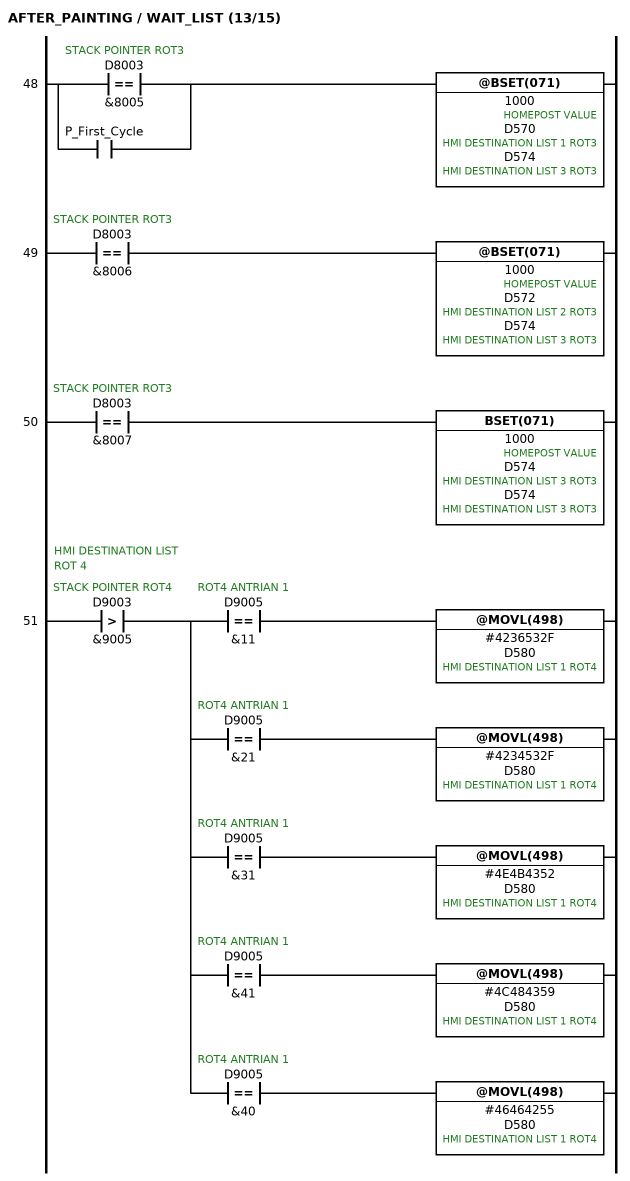
; [picture p96: AFTER_PAINTING / WAIT_LIST, rungs 48-51]
; rung 48
LD=(300) D8003 &8005  ; STACK POINTER ROT3
OR P_First_Cycle
@BSET(071) 1000 D570 D574  ; HOMEPOST VALUE, HMI DESTINATION LIST 1 ROT3, HMI DESTINATION LIST 3 ROT3
; rung 49
LD=(300) D8003 &8006  ; STACK POINTER ROT3
@BSET(071) 1000 D572 D574  ; HOMEPOST VALUE, HMI DESTINATION LIST 2 ROT3, HMI DESTINATION LIST 3 ROT3
; rung 50
LD=(300) D8003 &8007  ; STACK POINTER ROT3
BSET(071) 1000 D574 D574  ; HOMEPOST VALUE, HMI DESTINATION LIST 3 ROT3
; rung 51: HMI DESTINATION LIST / ROT 4
LD>(320) D9003 &9005  ; STACK POINTER ROT4
OUT TR0
AND=(300) D9005 &11  ; ROT4 ANTRIAN 1
@MOVL(498) #4236532F D580  ; HMI DESTINATION LIST 1 ROT4
LD TR0
AND=(300) D9005 &21  ; ROT4 ANTRIAN 1
@MOVL(498) #4234532F D580  ; HMI DESTINATION LIST 1 ROT4
LD TR0
AND=(300) D9005 &31  ; ROT4 ANTRIAN 1
@MOVL(498) #4E4B4352 D580  ; HMI DESTINATION LIST 1 ROT4
LD TR0
AND=(300) D9005 &41  ; ROT4 ANTRIAN 1
@MOVL(498) #4C484359 D580  ; HMI DESTINATION LIST 1 ROT4
LD TR0
AND=(300) D9005 &40  ; ROT4 ANTRIAN 1
@MOVL(498) #46464255 D580  ; HMI DESTINATION LIST 1 ROT4

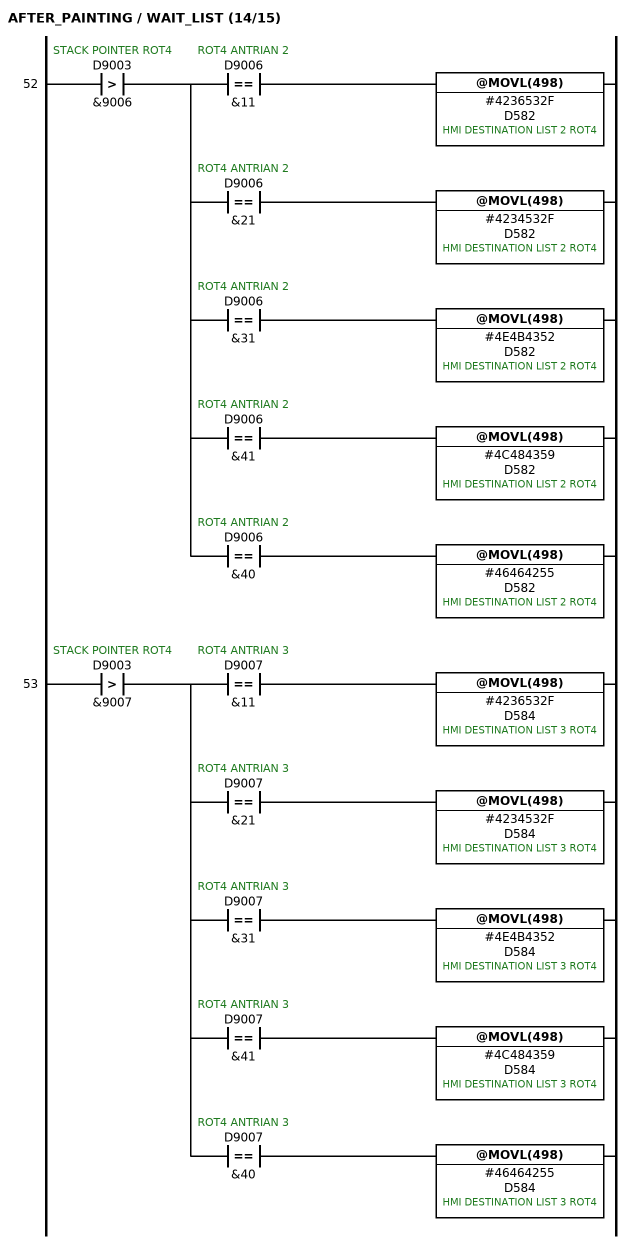
; rung 52
LD>(320) D9003 &9006  ; STACK POINTER ROT4
OUT TR0
AND=(300) D9006 &11  ; ROT4 ANTRIAN 2
@MOVL(498) #4236532F D582  ; HMI DESTINATION LIST 2 ROT4
LD TR0
AND=(300) D9006 &21  ; ROT4 ANTRIAN 2
@MOVL(498) #4234532F D582  ; HMI DESTINATION LIST 2 ROT4
LD TR0
AND=(300) D9006 &31  ; ROT4 ANTRIAN 2
@MOVL(498) #4E4B4352 D582  ; HMI DESTINATION LIST 2 ROT4
LD TR0
AND=(300) D9006 &41  ; ROT4 ANTRIAN 2
@MOVL(498) #4C484359 D582  ; HMI DESTINATION LIST 2 ROT4
LD TR0
AND=(300) D9006 &40  ; ROT4 ANTRIAN 2
@MOVL(498) #46464255 D582  ; HMI DESTINATION LIST 2 ROT4
; rung 53
LD>(320) D9003 &9007  ; STACK POINTER ROT4
OUT TR0
AND=(300) D9007 &11  ; ROT4 ANTRIAN 3
@MOVL(498) #4236532F D584  ; HMI DESTINATION LIST 3 ROT4
LD TR0
AND=(300) D9007 &21  ; ROT4 ANTRIAN 3
@MOVL(498) #4234532F D584  ; HMI DESTINATION LIST 3 ROT4
LD TR0
AND=(300) D9007 &31  ; ROT4 ANTRIAN 3
@MOVL(498) #4E4B4352 D584  ; HMI DESTINATION LIST 3 ROT4
LD TR0
AND=(300) D9007 &41  ; ROT4 ANTRIAN 3
@MOVL(498) #4C484359 D584  ; HMI DESTINATION LIST 3 ROT4
LD TR0
AND=(300) D9007 &40  ; ROT4 ANTRIAN 3
@MOVL(498) #46464255 D584  ; HMI DESTINATION LIST 3 ROT4

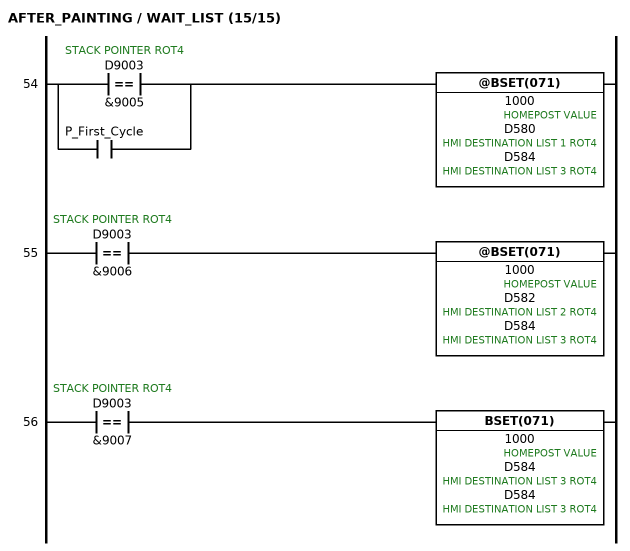
; rung 54
LD=(300) D9003 &9005  ; STACK POINTER ROT4
OR P_First_Cycle
@BSET(071) 1000 D580 D584  ; HOMEPOST VALUE, HMI DESTINATION LIST 1 ROT4, HMI DESTINATION LIST 3 ROT4
; rung 55
LD=(300) D9003 &9006  ; STACK POINTER ROT4
@BSET(071) 1000 D582 D584  ; HOMEPOST VALUE, HMI DESTINATION LIST 2 ROT4, HMI DESTINATION LIST 3 ROT4
; rung 56
LD=(300) D9003 &9007  ; STACK POINTER ROT4
BSET(071) 1000 D584 D584  ; HOMEPOST VALUE, HMI DESTINATION LIST 3 ROT4

### Section END
; rung 0
END(001)

## Function block MANUAL_ROTARY
VAR_INPUT
  PB_HMI_TURN : BOOL;
  PB_HMI_STRAIGHT : BOOL;
  PB_EXECUTE : BOOL;
  RS_PINLOCK_UP : BOOL;
  RS_PINLOCK_DOWN : BOOL;
  LS_STRAIGHT : BOOL;
  LS_TURN : BOOL;
  HOMEPOST_STRAIGHT : BOOL;
  HOMEPOST_RESET : BOOL;
END_VAR
VAR_OUTPUT
  MOTOR_FWD : BOOL;
  MOTOR_RVS : BOOL;
  PINLOCK_UP : BOOL;
  PINLOCK_DOWN : BOOL;
END_VAR
VAR
  MOTOR_RVS_MANUAL : BOOL;
  MOTOR_RVS_HOMEPOST : BOOL;
  PINLOCK_UP_STRAIGHT : BOOL;
  PINLOCK_UP_TURN : BOOL;
  PINLOCK_DOWN_STRAIGHT : BOOL;
  PINLOCK_DOWN_TURN : BOOL;
  PINLOCK_UP_HOMEPOST : BOOL;
  PINLOCK_DOWN_HOMEPOST : BOOL;
END_VAR

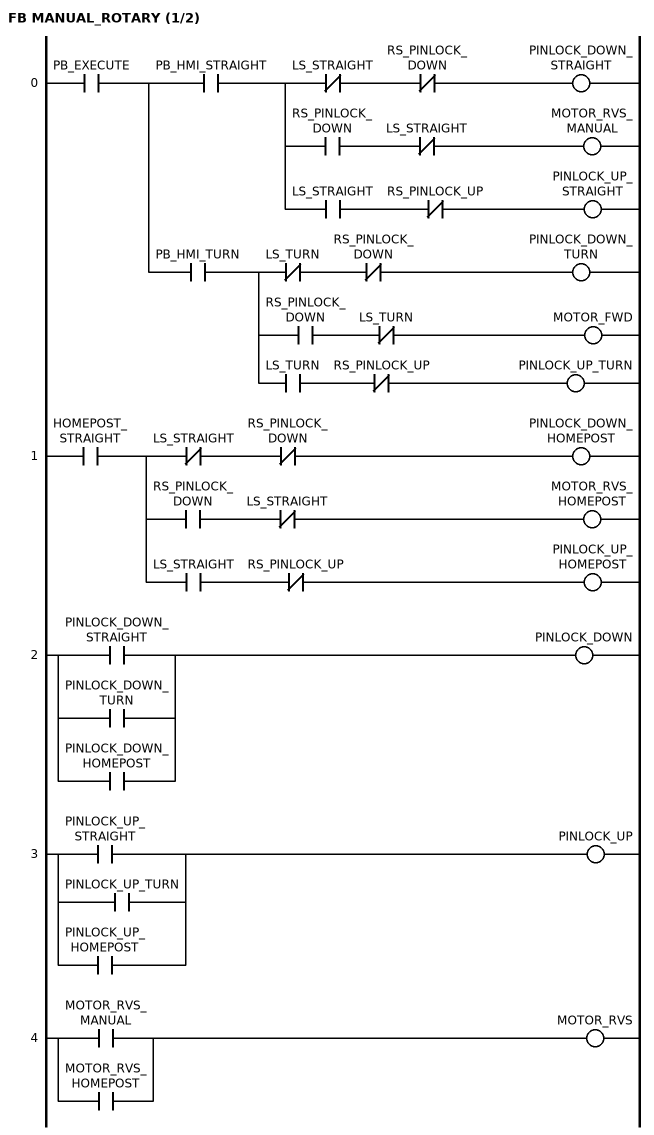
; rung 0
LD PB_EXECUTE
OUT TR0
AND PB_HMI_STRAIGHT
OUT TR1
ANDNOT LS_STRAIGHT
ANDNOT RS_PINLOCK_DOWN
OUT PINLOCK_DOWN_STRAIGHT
LD TR1
AND RS_PINLOCK_DOWN
ANDNOT LS_STRAIGHT
OUT MOTOR_RVS_MANUAL
LD TR1
AND LS_STRAIGHT
ANDNOT RS_PINLOCK_UP
OUT PINLOCK_UP_STRAIGHT
LD TR0
AND PB_HMI_TURN
OUT TR2
ANDNOT LS_TURN
ANDNOT RS_PINLOCK_DOWN
OUT PINLOCK_DOWN_TURN
LD TR2
AND RS_PINLOCK_DOWN
ANDNOT LS_TURN
OUT MOTOR_FWD
LD TR2
AND LS_TURN
ANDNOT RS_PINLOCK_UP
OUT PINLOCK_UP_TURN
; rung 1
LD HOMEPOST_STRAIGHT
OUT TR0
ANDNOT LS_STRAIGHT
ANDNOT RS_PINLOCK_DOWN
OUT PINLOCK_DOWN_HOMEPOST
LD TR0
AND RS_PINLOCK_DOWN
ANDNOT LS_STRAIGHT
OUT MOTOR_RVS_HOMEPOST
LD TR0
AND LS_STRAIGHT
ANDNOT RS_PINLOCK_UP
OUT PINLOCK_UP_HOMEPOST
; rung 2
LD PINLOCK_DOWN_STRAIGHT
OR PINLOCK_DOWN_TURN
OR PINLOCK_DOWN_HOMEPOST
OUT PINLOCK_DOWN
; rung 3
LD PINLOCK_UP_STRAIGHT
OR PINLOCK_UP_TURN
OR PINLOCK_UP_HOMEPOST
OUT PINLOCK_UP
; rung 4
LD MOTOR_RVS_MANUAL
OR MOTOR_RVS_HOMEPOST
OUT MOTOR_RVS

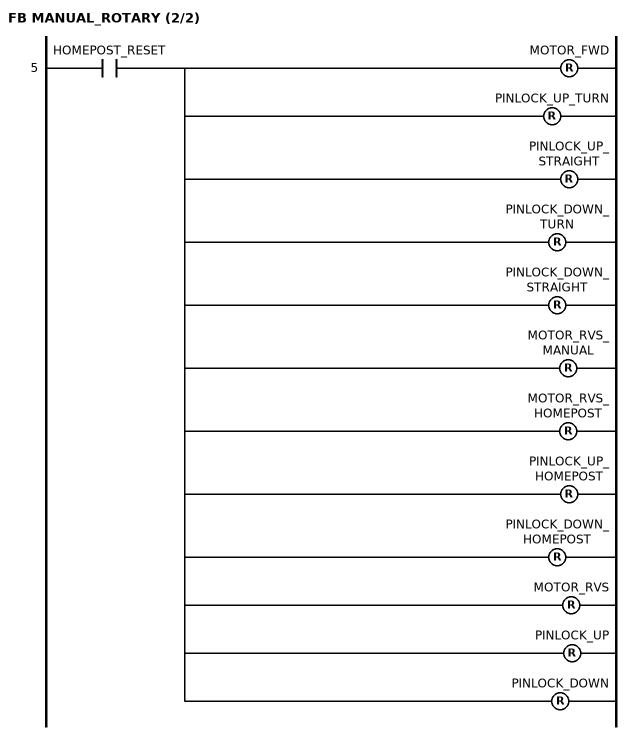
; rung 5
LD HOMEPOST_RESET
RSET MOTOR_FWD
RSET PINLOCK_UP_TURN
RSET PINLOCK_UP_STRAIGHT
RSET PINLOCK_DOWN_TURN
RSET PINLOCK_DOWN_STRAIGHT
RSET MOTOR_RVS_MANUAL
RSET MOTOR_RVS_HOMEPOST
RSET PINLOCK_UP_HOMEPOST
RSET PINLOCK_DOWN_HOMEPOST
RSET MOTOR_RVS
RSET PINLOCK_UP
RSET PINLOCK_DOWN

## Function block RFID_SEQUENCE
VAR_INPUT
  PB_SAVE : BOOL;
  AUTO_SEQ_ON : BOOL;
  INPUT_DATA : UINT;
  PH_OUT : BOOL;
  MANUAL_MODE : BOOL;
  PB_CLEAR_MEMORY : BOOL;
  PB_ENABLE_READER : BOOL;
  OUT_HMI_DISPLAY_NO_RFID : UDINT;
  STACK_LOC : UINT;
  REDUDANCY_ACCEPTED : BOOL;
  HOMEPOST_RESET : BOOL;
END_VAR
VAR_OUTPUT
  RFID_CONFIRM_MATCH : BOOL;
  DISPLAY_TEACH_RFID : UDINT;
  ALARM_RFID_NOT_DETECT : BOOL;
  DATA_REDUDANCY : BOOL;
  RETAIN MEMORY_1 : UDINT;
  RETAIN MEMORY_2 : UDINT;
  RETAIN MEMORY_3 : UDINT;
  RETAIN MEMORY_4 : UDINT;
  RETAIN MEMORY_5 : UDINT;
  RETAIN MEMORY_6 : UDINT;
  RETAIN MEMORY_7 : UDINT;
  RETAIN MEMORY_8 : UDINT;
  RETAIN MEMORY_9 : UDINT;
  RETAIN MEMORY_10 : UDINT;
  RETAIN MEMORY_11 : UDINT;
  RETAIN MEMORY_12 : UDINT;
  RETAIN MEMORY_13 : UDINT;
  RETAIN MEMORY_14 : UDINT;
  RETAIN MEMORY_15 : UDINT;
  RETAIN MEMORY_16 : UDINT;
  RETAIN MEMORY_17 : UDINT;
  RETAIN MEMORY_18 : UDINT;
  RETAIN MEMORY_19 : UDINT;
  RETAIN MEMORY_20 : UDINT;
  RETAIN MEMORY_21 : UDINT;
  RETAIN MEMORY_22 : UDINT;
  RETAIN MEMORY_23 : UDINT;
  RETAIN MEMORY_24 : UDINT;
  RETAIN MEMORY_25 : UDINT;
  RETAIN MEMORY_26 : UDINT;
  RETAIN MEMORY_27 : UDINT;
  RETAIN MEMORY_28 : UDINT;
  RETAIN MEMORY_29 : UDINT;
  RETAIN MEMORY_30 : UDINT;
  RETAIN MEMORY_31 : UDINT;
  RETAIN MEMORY_32 : UDINT;
  RETAIN MEMORY_33 : UDINT;
  RETAIN MEMORY_34 : UDINT;
  RETAIN MEMORY_35 : UDINT;
  RETAIN MEMORY_36 : UDINT;
  RETAIN MEMORY_37 : UDINT;
  RETAIN MEMORY_38 : UDINT;
  RETAIN MEMORY_39 : UDINT;
  RETAIN MEMORY_40 : UDINT;
  RETAIN MEMORY_41 : UDINT;
  RETAIN MEMORY_42 : UDINT;
  RETAIN MEMORY_43 : UDINT;
  RETAIN MEMORY_44 : UDINT;
  RETAIN MEMORY_45 : UDINT;
  RETAIN MEMORY_46 : UDINT;
  RETAIN MEMORY_47 : UDINT;
  RETAIN MEMORY_48 : UDINT;
  RETAIN MEMORY_49 : UDINT;
  RETAIN MEMORY_50 : UDINT;
END_VAR
VAR
  TIMER_RFID_READ_TIMEOUT : TIMER;
  TIMER_RFID_NOT_REGISTERED : TIMER;
END_VAR

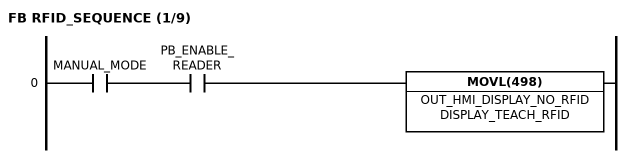
; rung 0
LD MANUAL_MODE
AND PB_ENABLE_READER
MOVL(498) OUT_HMI_DISPLAY_NO_RFID DISPLAY_TEACH_RFID

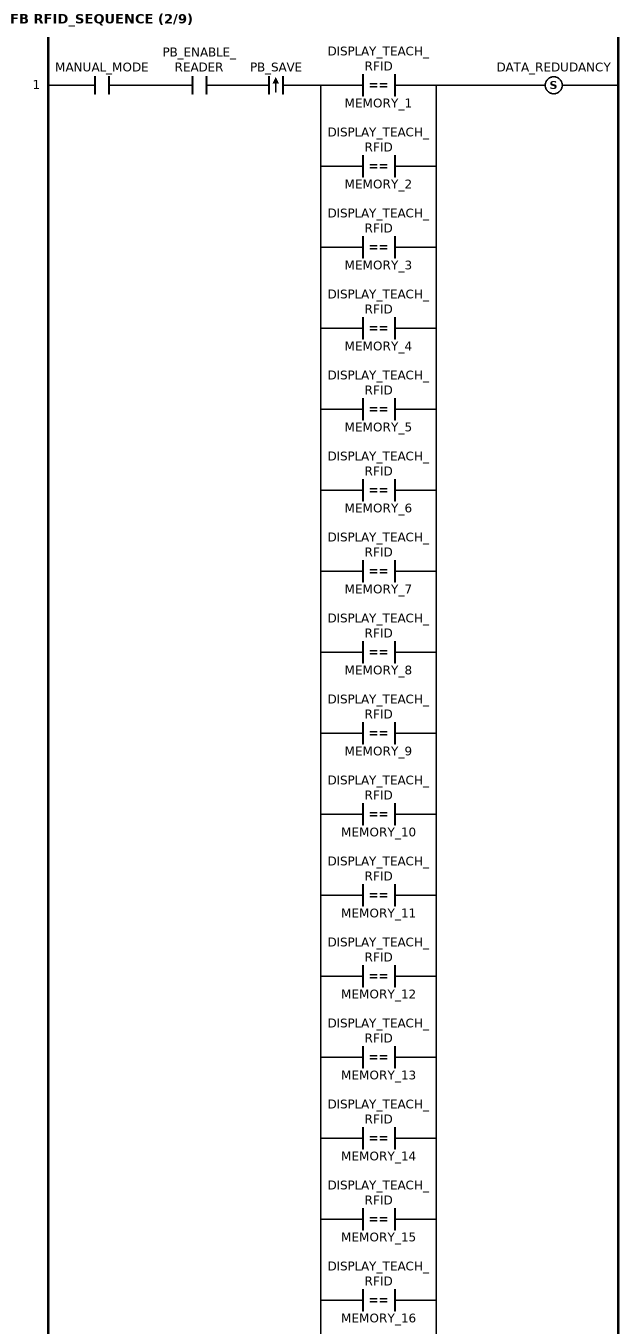

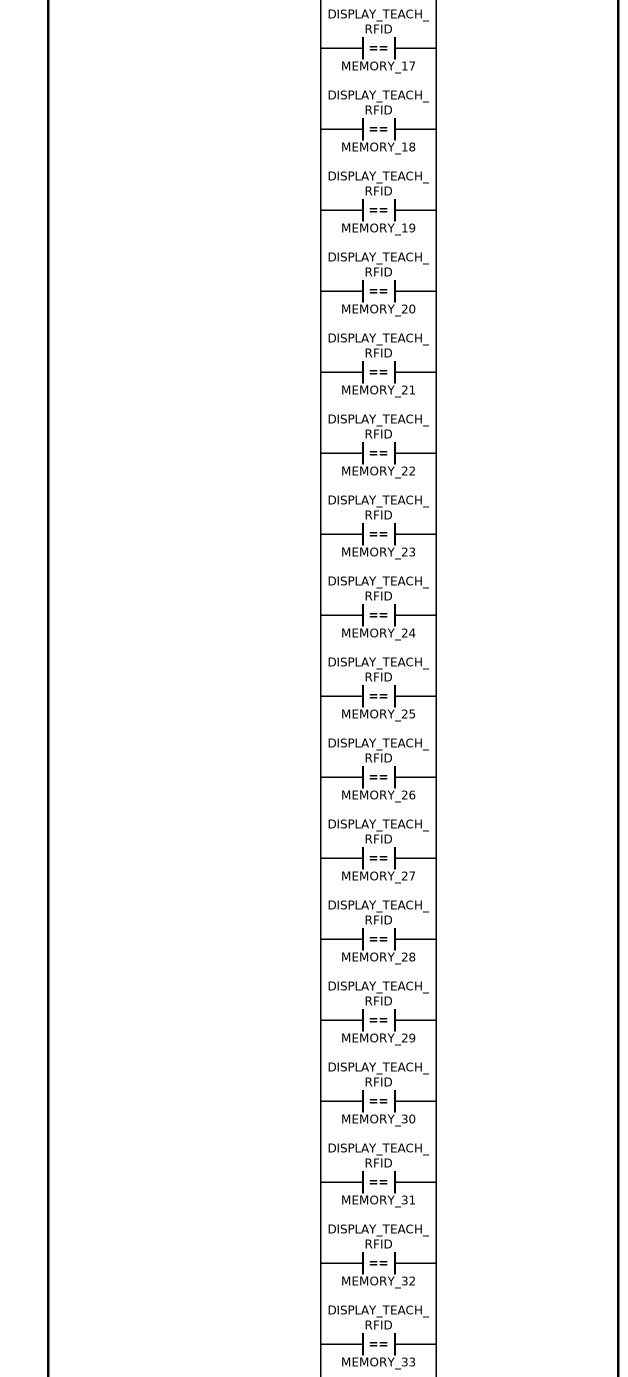

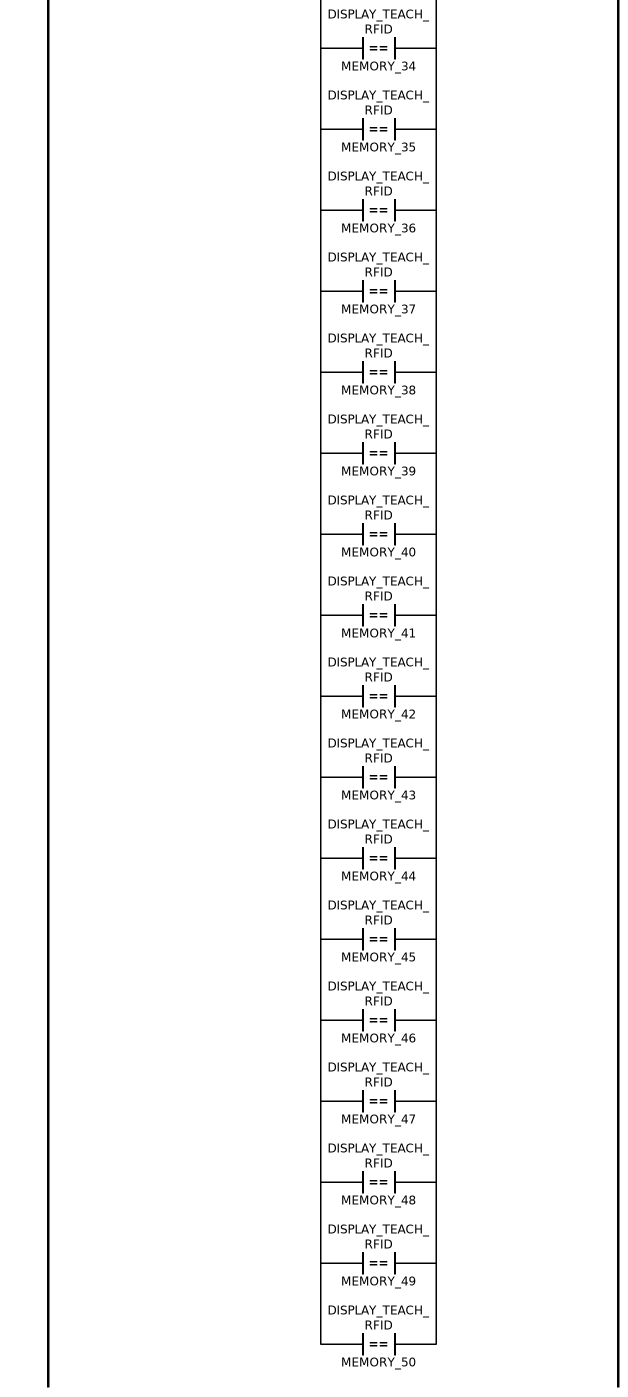
; rung 1
LD MANUAL_MODE
AND PB_ENABLE_READER
@AND PB_SAVE
LD=(300) DISPLAY_TEACH_RFID MEMORY_1
OR=(300) DISPLAY_TEACH_RFID MEMORY_2
OR=(300) DISPLAY_TEACH_RFID MEMORY_3
OR=(300) DISPLAY_TEACH_RFID MEMORY_4
OR=(300) DISPLAY_TEACH_RFID MEMORY_5
OR=(300) DISPLAY_TEACH_RFID MEMORY_6
OR=(300) DISPLAY_TEACH_RFID MEMORY_7
OR=(300) DISPLAY_TEACH_RFID MEMORY_8
OR=(300) DISPLAY_TEACH_RFID MEMORY_9
OR=(300) DISPLAY_TEACH_RFID MEMORY_10
OR=(300) DISPLAY_TEACH_RFID MEMORY_11
OR=(300) DISPLAY_TEACH_RFID MEMORY_12
OR=(300) DISPLAY_TEACH_RFID MEMORY_13
OR=(300) DISPLAY_TEACH_RFID MEMORY_14
OR=(300) DISPLAY_TEACH_RFID MEMORY_15
OR=(300) DISPLAY_TEACH_RFID MEMORY_16
OR=(300) DISPLAY_TEACH_RFID MEMORY_17
OR=(300) DISPLAY_TEACH_RFID MEMORY_18
OR=(300) DISPLAY_TEACH_RFID MEMORY_19
OR=(300) DISPLAY_TEACH_RFID MEMORY_20
OR=(300) DISPLAY_TEACH_RFID MEMORY_21
OR=(300) DISPLAY_TEACH_RFID MEMORY_22
OR=(300) DISPLAY_TEACH_RFID MEMORY_23
OR=(300) DISPLAY_TEACH_RFID MEMORY_24
OR=(300) DISPLAY_TEACH_RFID MEMORY_25
OR=(300) DISPLAY_TEACH_RFID MEMORY_26
OR=(300) DISPLAY_TEACH_RFID MEMORY_27
OR=(300) DISPLAY_TEACH_RFID MEMORY_28
OR=(300) DISPLAY_TEACH_RFID MEMORY_29
OR=(300) DISPLAY_TEACH_RFID MEMORY_30
OR=(300) DISPLAY_TEACH_RFID MEMORY_31
OR=(300) DISPLAY_TEACH_RFID MEMORY_32
OR=(300) DISPLAY_TEACH_RFID MEMORY_33
OR=(300) DISPLAY_TEACH_RFID MEMORY_34
OR=(300) DISPLAY_TEACH_RFID MEMORY_35
OR=(300) DISPLAY_TEACH_RFID MEMORY_36
OR=(300) DISPLAY_TEACH_RFID MEMORY_37
OR=(300) DISPLAY_TEACH_RFID MEMORY_38
OR=(300) DISPLAY_TEACH_RFID MEMORY_39
OR=(300) DISPLAY_TEACH_RFID MEMORY_40
OR=(300) DISPLAY_TEACH_RFID MEMORY_41
OR=(300) DISPLAY_TEACH_RFID MEMORY_42
OR=(300) DISPLAY_TEACH_RFID MEMORY_43
OR=(300) DISPLAY_TEACH_RFID MEMORY_44
OR=(300) DISPLAY_TEACH_RFID MEMORY_45
OR=(300) DISPLAY_TEACH_RFID MEMORY_46
OR=(300) DISPLAY_TEACH_RFID MEMORY_47
OR=(300) DISPLAY_TEACH_RFID MEMORY_48
OR=(300) DISPLAY_TEACH_RFID MEMORY_49
OR=(300) DISPLAY_TEACH_RFID MEMORY_50
ANDLD
SET DATA_REDUDANCY

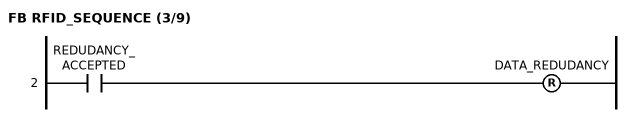
; rung 2
LD REDUDANCY_ACCEPTED
RSET DATA_REDUDANCY

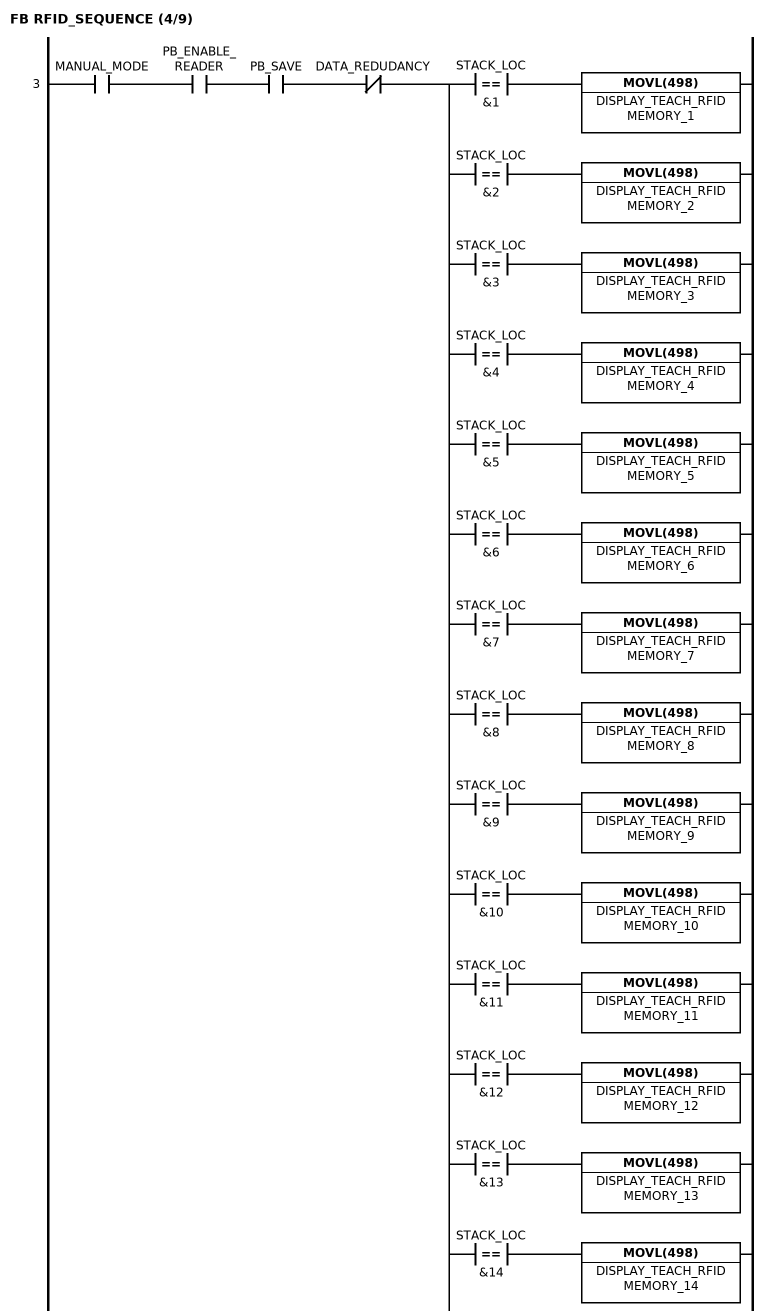

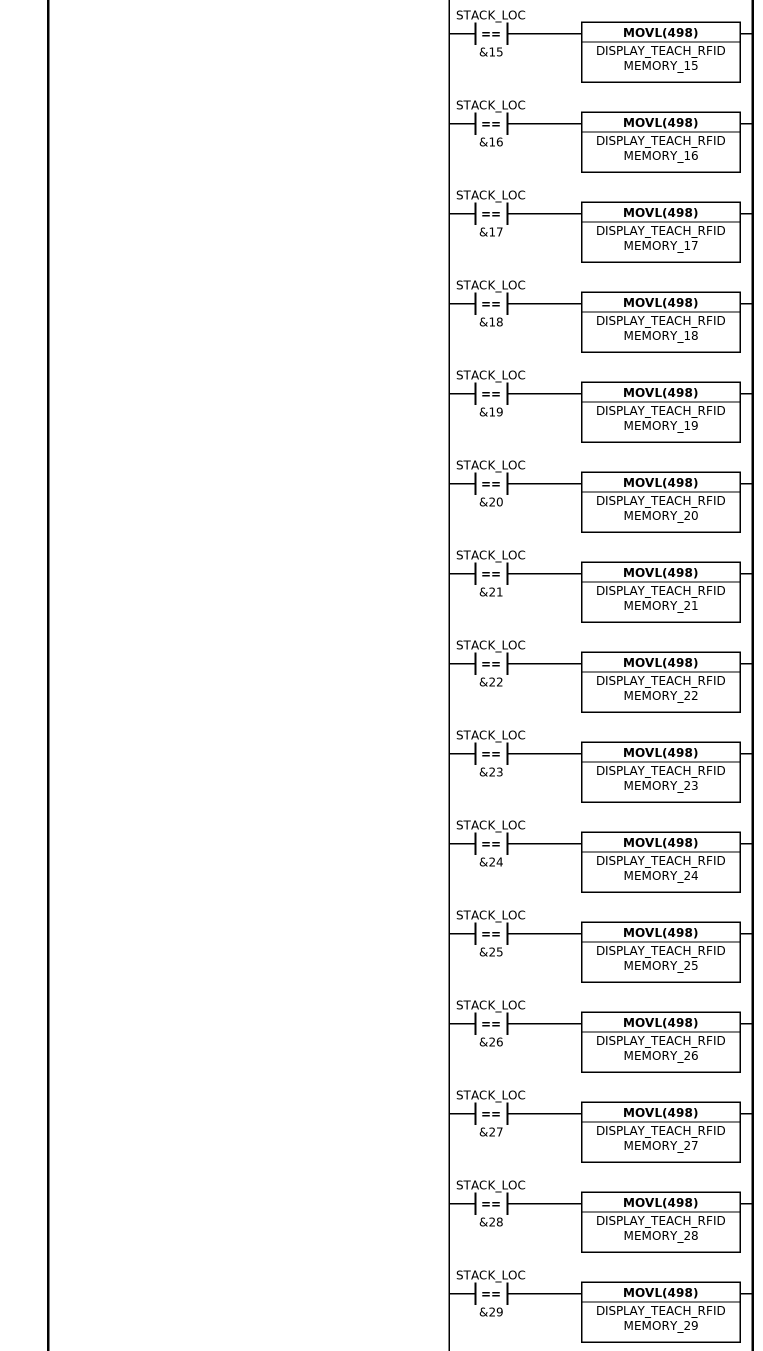

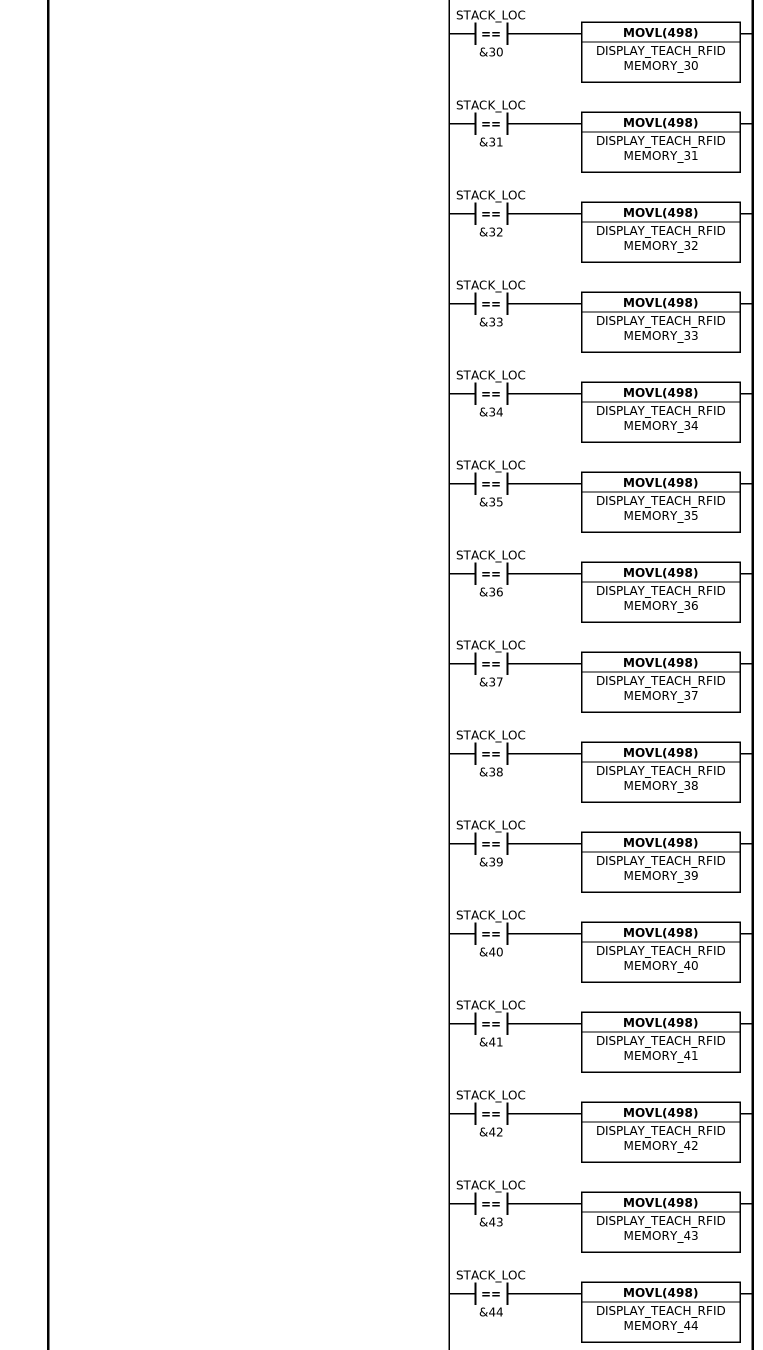

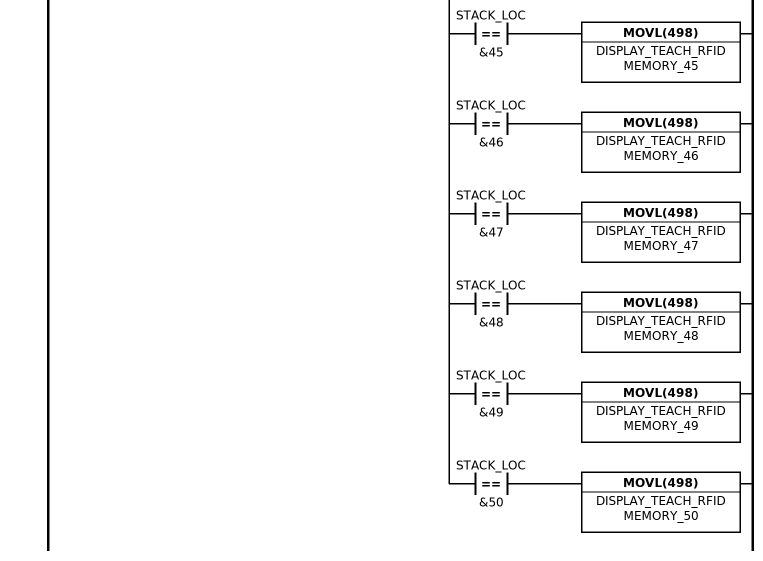
; rung 3
LD MANUAL_MODE
AND PB_ENABLE_READER
AND PB_SAVE
ANDNOT DATA_REDUDANCY
OUT TR0
AND=(300) STACK_LOC &1
MOVL(498) DISPLAY_TEACH_RFID MEMORY_1
LD TR0
AND=(300) STACK_LOC &2
MOVL(498) DISPLAY_TEACH_RFID MEMORY_2
LD TR0
AND=(300) STACK_LOC &3
MOVL(498) DISPLAY_TEACH_RFID MEMORY_3
LD TR0
AND=(300) STACK_LOC &4
MOVL(498) DISPLAY_TEACH_RFID MEMORY_4
LD TR0
AND=(300) STACK_LOC &5
MOVL(498) DISPLAY_TEACH_RFID MEMORY_5
LD TR0
AND=(300) STACK_LOC &6
MOVL(498) DISPLAY_TEACH_RFID MEMORY_6
LD TR0
AND=(300) STACK_LOC &7
MOVL(498) DISPLAY_TEACH_RFID MEMORY_7
LD TR0
AND=(300) STACK_LOC &8
MOVL(498) DISPLAY_TEACH_RFID MEMORY_8
LD TR0
AND=(300) STACK_LOC &9
MOVL(498) DISPLAY_TEACH_RFID MEMORY_9
LD TR0
AND=(300) STACK_LOC &10
MOVL(498) DISPLAY_TEACH_RFID MEMORY_10
LD TR0
AND=(300) STACK_LOC &11
MOVL(498) DISPLAY_TEACH_RFID MEMORY_11
LD TR0
AND=(300) STACK_LOC &12
MOVL(498) DISPLAY_TEACH_RFID MEMORY_12
LD TR0
AND=(300) STACK_LOC &13
MOVL(498) DISPLAY_TEACH_RFID MEMORY_13
LD TR0
AND=(300) STACK_LOC &14
MOVL(498) DISPLAY_TEACH_RFID MEMORY_14
LD TR0
AND=(300) STACK_LOC &15
MOVL(498) DISPLAY_TEACH_RFID MEMORY_15
LD TR0
AND=(300) STACK_LOC &16
MOVL(498) DISPLAY_TEACH_RFID MEMORY_16
LD TR0
AND=(300) STACK_LOC &17
MOVL(498) DISPLAY_TEACH_RFID MEMORY_17
LD TR0
AND=(300) STACK_LOC &18
MOVL(498) DISPLAY_TEACH_RFID MEMORY_18
LD TR0
AND=(300) STACK_LOC &19
MOVL(498) DISPLAY_TEACH_RFID MEMORY_19
LD TR0
AND=(300) STACK_LOC &20
MOVL(498) DISPLAY_TEACH_RFID MEMORY_20
LD TR0
AND=(300) STACK_LOC &21
MOVL(498) DISPLAY_TEACH_RFID MEMORY_21
LD TR0
AND=(300) STACK_LOC &22
MOVL(498) DISPLAY_TEACH_RFID MEMORY_22
LD TR0
AND=(300) STACK_LOC &23
MOVL(498) DISPLAY_TEACH_RFID MEMORY_23
LD TR0
AND=(300) STACK_LOC &24
MOVL(498) DISPLAY_TEACH_RFID MEMORY_24
LD TR0
AND=(300) STACK_LOC &25
MOVL(498) DISPLAY_TEACH_RFID MEMORY_25
LD TR0
AND=(300) STACK_LOC &26
MOVL(498) DISPLAY_TEACH_RFID MEMORY_26
LD TR0
AND=(300) STACK_LOC &27
MOVL(498) DISPLAY_TEACH_RFID MEMORY_27
LD TR0
AND=(300) STACK_LOC &28
MOVL(498) DISPLAY_TEACH_RFID MEMORY_28
LD TR0
AND=(300) STACK_LOC &29
MOVL(498) DISPLAY_TEACH_RFID MEMORY_29
LD TR0
AND=(300) STACK_LOC &30
MOVL(498) DISPLAY_TEACH_RFID MEMORY_30
LD TR0
AND=(300) STACK_LOC &31
MOVL(498) DISPLAY_TEACH_RFID MEMORY_31
LD TR0
AND=(300) STACK_LOC &32
MOVL(498) DISPLAY_TEACH_RFID MEMORY_32
LD TR0
AND=(300) STACK_LOC &33
MOVL(498) DISPLAY_TEACH_RFID MEMORY_33
LD TR0
AND=(300) STACK_LOC &34
MOVL(498) DISPLAY_TEACH_RFID MEMORY_34
LD TR0
AND=(300) STACK_LOC &35
MOVL(498) DISPLAY_TEACH_RFID MEMORY_35
LD TR0
AND=(300) STACK_LOC &36
MOVL(498) DISPLAY_TEACH_RFID MEMORY_36
LD TR0
AND=(300) STACK_LOC &37
MOVL(498) DISPLAY_TEACH_RFID MEMORY_37
LD TR0
AND=(300) STACK_LOC &38
MOVL(498) DISPLAY_TEACH_RFID MEMORY_38
LD TR0
AND=(300) STACK_LOC &39
MOVL(498) DISPLAY_TEACH_RFID MEMORY_39
LD TR0
AND=(300) STACK_LOC &40
MOVL(498) DISPLAY_TEACH_RFID MEMORY_40
LD TR0
AND=(300) STACK_LOC &41
MOVL(498) DISPLAY_TEACH_RFID MEMORY_41
LD TR0
AND=(300) STACK_LOC &42
MOVL(498) DISPLAY_TEACH_RFID MEMORY_42
LD TR0
AND=(300) STACK_LOC &43
MOVL(498) DISPLAY_TEACH_RFID MEMORY_43
LD TR0
AND=(300) STACK_LOC &44
MOVL(498) DISPLAY_TEACH_RFID MEMORY_44
LD TR0
AND=(300) STACK_LOC &45
MOVL(498) DISPLAY_TEACH_RFID MEMORY_45
LD TR0
AND=(300) STACK_LOC &46
MOVL(498) DISPLAY_TEACH_RFID MEMORY_46
LD TR0
AND=(300) STACK_LOC &47
MOVL(498) DISPLAY_TEACH_RFID MEMORY_47
LD TR0
AND=(300) STACK_LOC &48
MOVL(498) DISPLAY_TEACH_RFID MEMORY_48
LD TR0
AND=(300) STACK_LOC &49
MOVL(498) DISPLAY_TEACH_RFID MEMORY_49
LD TR0
AND=(300) STACK_LOC &50
MOVL(498) DISPLAY_TEACH_RFID MEMORY_50

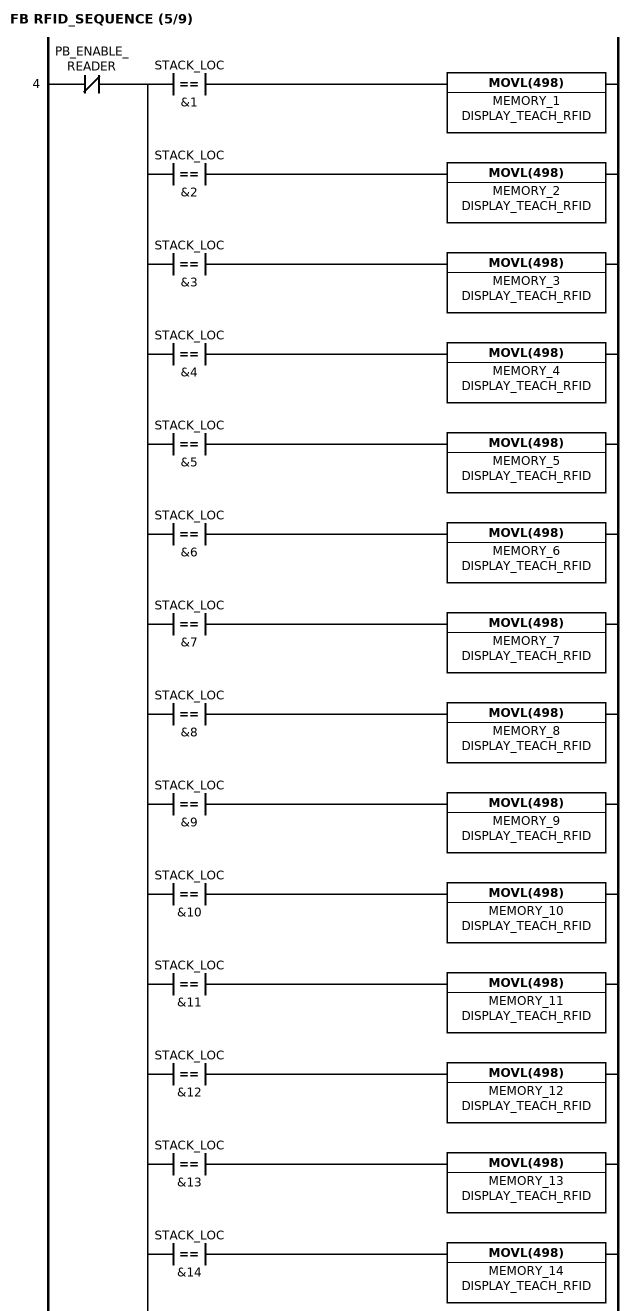

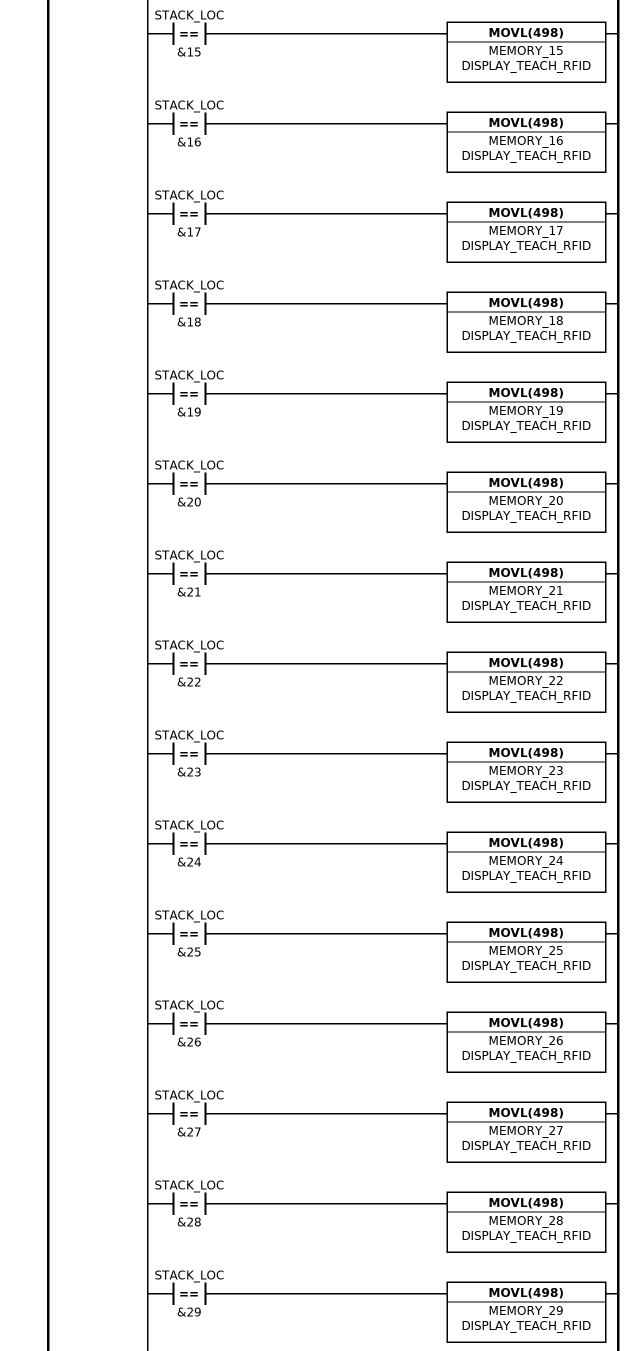

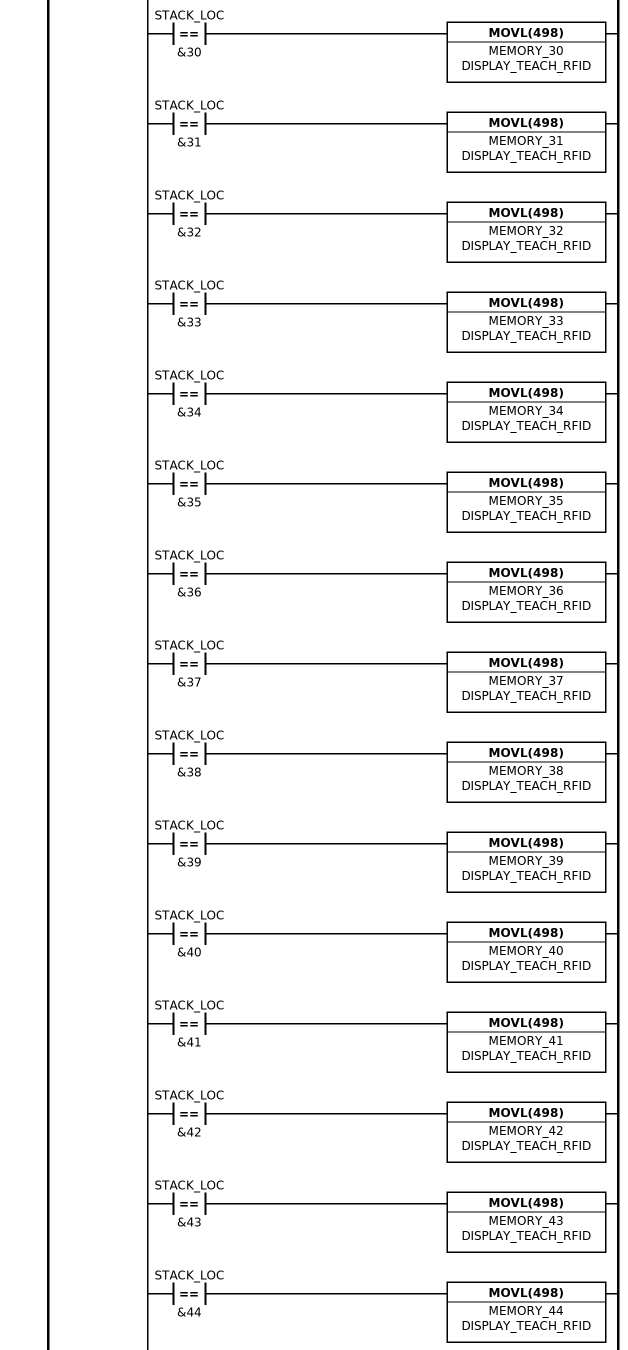

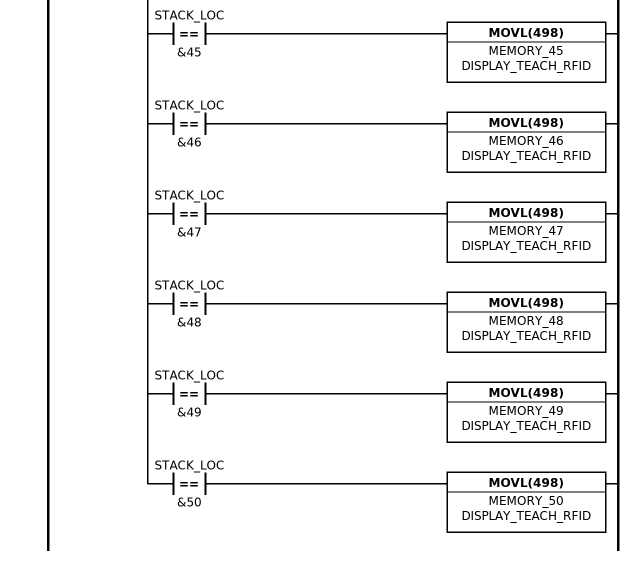
; rung 4
LDNOT PB_ENABLE_READER
OUT TR0
AND=(300) STACK_LOC &1
MOVL(498) MEMORY_1 DISPLAY_TEACH_RFID
LD TR0
AND=(300) STACK_LOC &2
MOVL(498) MEMORY_2 DISPLAY_TEACH_RFID
LD TR0
AND=(300) STACK_LOC &3
MOVL(498) MEMORY_3 DISPLAY_TEACH_RFID
LD TR0
AND=(300) STACK_LOC &4
MOVL(498) MEMORY_4 DISPLAY_TEACH_RFID
LD TR0
AND=(300) STACK_LOC &5
MOVL(498) MEMORY_5 DISPLAY_TEACH_RFID
LD TR0
AND=(300) STACK_LOC &6
MOVL(498) MEMORY_6 DISPLAY_TEACH_RFID
LD TR0
AND=(300) STACK_LOC &7
MOVL(498) MEMORY_7 DISPLAY_TEACH_RFID
LD TR0
AND=(300) STACK_LOC &8
MOVL(498) MEMORY_8 DISPLAY_TEACH_RFID
LD TR0
AND=(300) STACK_LOC &9
MOVL(498) MEMORY_9 DISPLAY_TEACH_RFID
LD TR0
AND=(300) STACK_LOC &10
MOVL(498) MEMORY_10 DISPLAY_TEACH_RFID
LD TR0
AND=(300) STACK_LOC &11
MOVL(498) MEMORY_11 DISPLAY_TEACH_RFID
LD TR0
AND=(300) STACK_LOC &12
MOVL(498) MEMORY_12 DISPLAY_TEACH_RFID
LD TR0
AND=(300) STACK_LOC &13
MOVL(498) MEMORY_13 DISPLAY_TEACH_RFID
LD TR0
AND=(300) STACK_LOC &14
MOVL(498) MEMORY_14 DISPLAY_TEACH_RFID
LD TR0
AND=(300) STACK_LOC &15
MOVL(498) MEMORY_15 DISPLAY_TEACH_RFID
LD TR0
AND=(300) STACK_LOC &16
MOVL(498) MEMORY_16 DISPLAY_TEACH_RFID
LD TR0
AND=(300) STACK_LOC &17
MOVL(498) MEMORY_17 DISPLAY_TEACH_RFID
LD TR0
AND=(300) STACK_LOC &18
MOVL(498) MEMORY_18 DISPLAY_TEACH_RFID
LD TR0
AND=(300) STACK_LOC &19
MOVL(498) MEMORY_19 DISPLAY_TEACH_RFID
LD TR0
AND=(300) STACK_LOC &20
MOVL(498) MEMORY_20 DISPLAY_TEACH_RFID
LD TR0
AND=(300) STACK_LOC &21
MOVL(498) MEMORY_21 DISPLAY_TEACH_RFID
LD TR0
AND=(300) STACK_LOC &22
MOVL(498) MEMORY_22 DISPLAY_TEACH_RFID
LD TR0
AND=(300) STACK_LOC &23
MOVL(498) MEMORY_23 DISPLAY_TEACH_RFID
LD TR0
AND=(300) STACK_LOC &24
MOVL(498) MEMORY_24 DISPLAY_TEACH_RFID
LD TR0
AND=(300) STACK_LOC &25
MOVL(498) MEMORY_25 DISPLAY_TEACH_RFID
LD TR0
AND=(300) STACK_LOC &26
MOVL(498) MEMORY_26 DISPLAY_TEACH_RFID
LD TR0
AND=(300) STACK_LOC &27
MOVL(498) MEMORY_27 DISPLAY_TEACH_RFID
LD TR0
AND=(300) STACK_LOC &28
MOVL(498) MEMORY_28 DISPLAY_TEACH_RFID
LD TR0
AND=(300) STACK_LOC &29
MOVL(498) MEMORY_29 DISPLAY_TEACH_RFID
LD TR0
AND=(300) STACK_LOC &30
MOVL(498) MEMORY_30 DISPLAY_TEACH_RFID
LD TR0
AND=(300) STACK_LOC &31
MOVL(498) MEMORY_31 DISPLAY_TEACH_RFID
LD TR0
AND=(300) STACK_LOC &32
MOVL(498) MEMORY_32 DISPLAY_TEACH_RFID
LD TR0
AND=(300) STACK_LOC &33
MOVL(498) MEMORY_33 DISPLAY_TEACH_RFID
LD TR0
AND=(300) STACK_LOC &34
MOVL(498) MEMORY_34 DISPLAY_TEACH_RFID
LD TR0
AND=(300) STACK_LOC &35
MOVL(498) MEMORY_35 DISPLAY_TEACH_RFID
LD TR0
AND=(300) STACK_LOC &36
MOVL(498) MEMORY_36 DISPLAY_TEACH_RFID
LD TR0
AND=(300) STACK_LOC &37
MOVL(498) MEMORY_37 DISPLAY_TEACH_RFID
LD TR0
AND=(300) STACK_LOC &38
MOVL(498) MEMORY_38 DISPLAY_TEACH_RFID
LD TR0
AND=(300) STACK_LOC &39
MOVL(498) MEMORY_39 DISPLAY_TEACH_RFID
LD TR0
AND=(300) STACK_LOC &40
MOVL(498) MEMORY_40 DISPLAY_TEACH_RFID
LD TR0
AND=(300) STACK_LOC &41
MOVL(498) MEMORY_41 DISPLAY_TEACH_RFID
LD TR0
AND=(300) STACK_LOC &42
MOVL(498) MEMORY_42 DISPLAY_TEACH_RFID
LD TR0
AND=(300) STACK_LOC &43
MOVL(498) MEMORY_43 DISPLAY_TEACH_RFID
LD TR0
AND=(300) STACK_LOC &44
MOVL(498) MEMORY_44 DISPLAY_TEACH_RFID
LD TR0
AND=(300) STACK_LOC &45
MOVL(498) MEMORY_45 DISPLAY_TEACH_RFID
LD TR0
AND=(300) STACK_LOC &46
MOVL(498) MEMORY_46 DISPLAY_TEACH_RFID
LD TR0
AND=(300) STACK_LOC &47
MOVL(498) MEMORY_47 DISPLAY_TEACH_RFID
LD TR0
AND=(300) STACK_LOC &48
MOVL(498) MEMORY_48 DISPLAY_TEACH_RFID
LD TR0
AND=(300) STACK_LOC &49
MOVL(498) MEMORY_49 DISPLAY_TEACH_RFID
LD TR0
AND=(300) STACK_LOC &50
MOVL(498) MEMORY_50 DISPLAY_TEACH_RFID

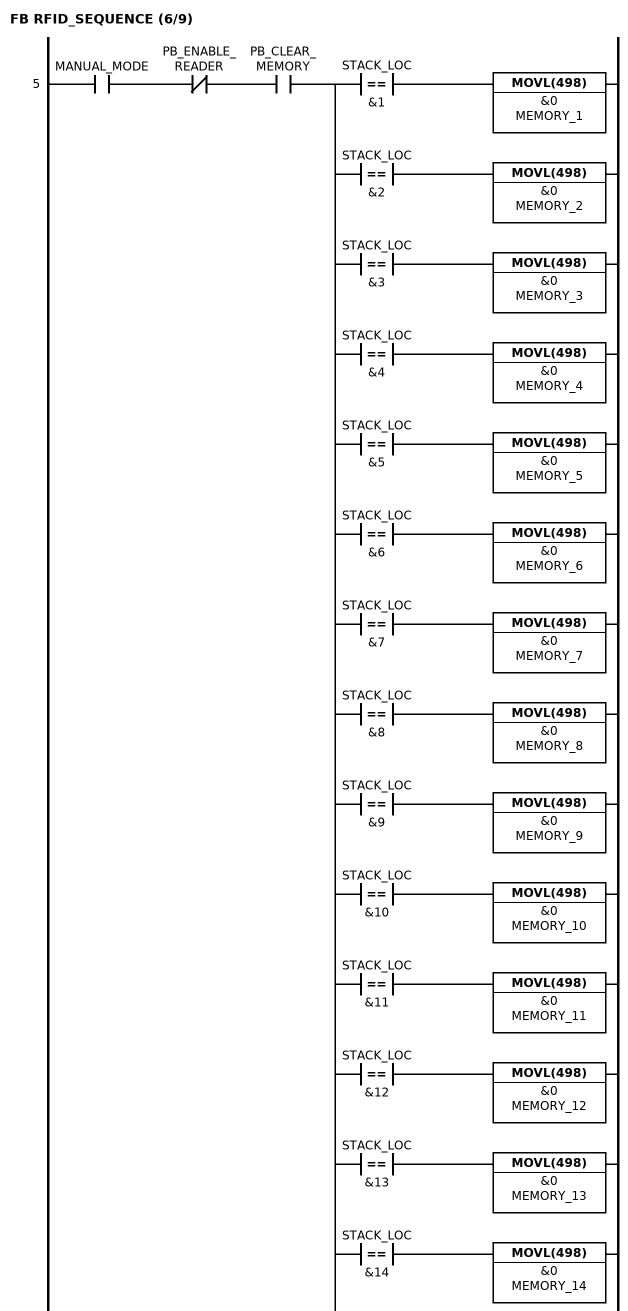

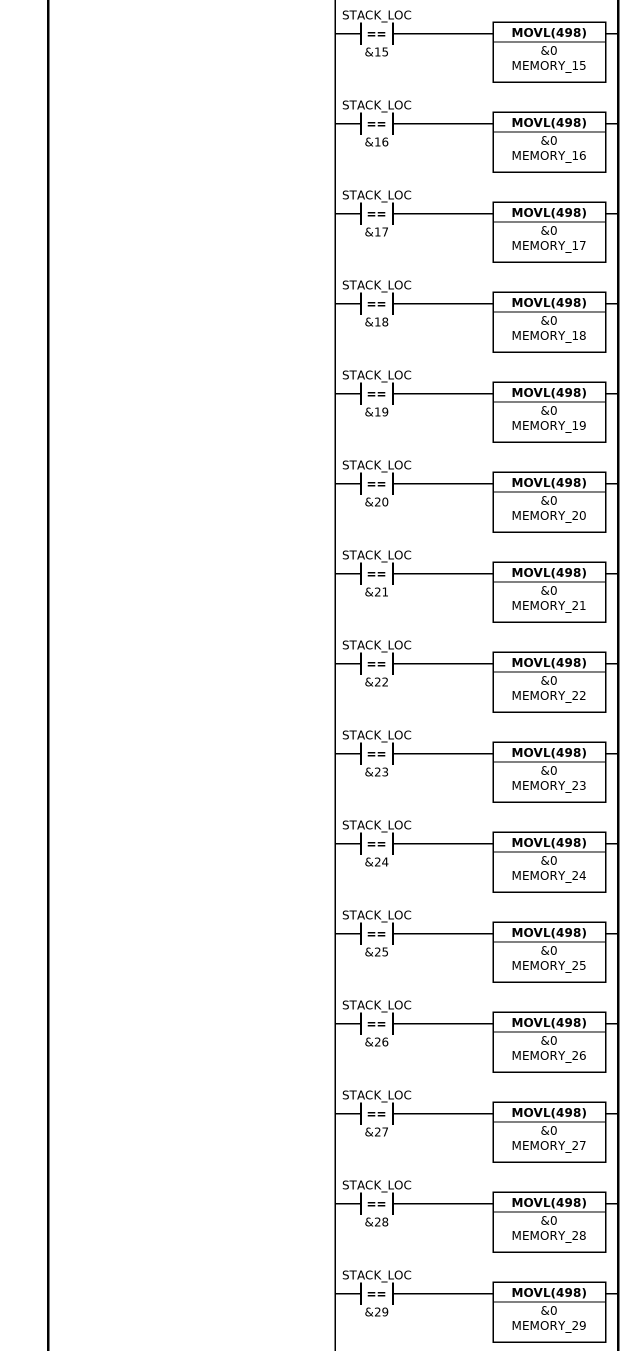

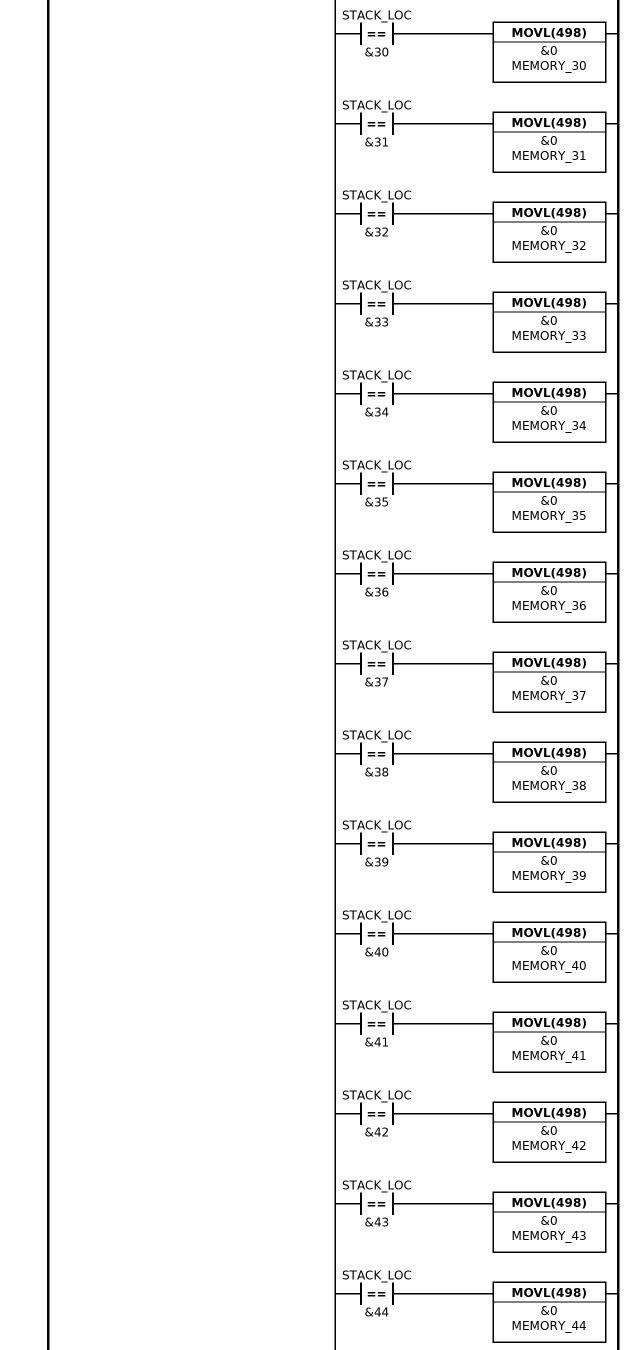

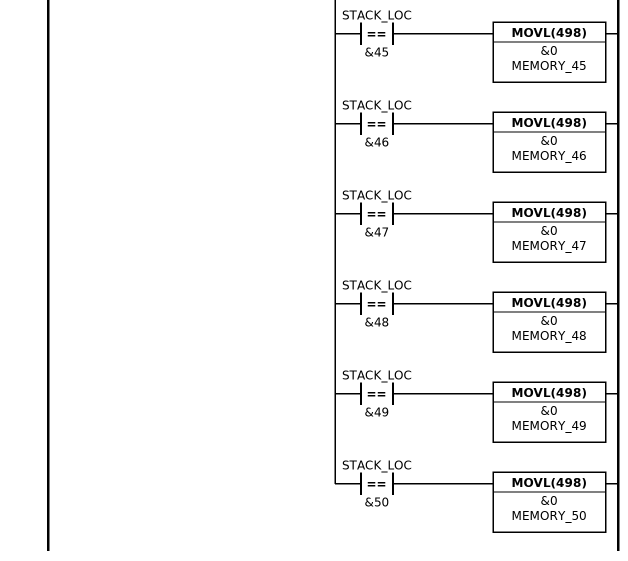
; rung 5
LD MANUAL_MODE
ANDNOT PB_ENABLE_READER
AND PB_CLEAR_MEMORY
OUT TR0
AND=(300) STACK_LOC &1
MOVL(498) &0 MEMORY_1
LD TR0
AND=(300) STACK_LOC &2
MOVL(498) &0 MEMORY_2
LD TR0
AND=(300) STACK_LOC &3
MOVL(498) &0 MEMORY_3
LD TR0
AND=(300) STACK_LOC &4
MOVL(498) &0 MEMORY_4
LD TR0
AND=(300) STACK_LOC &5
MOVL(498) &0 MEMORY_5
LD TR0
AND=(300) STACK_LOC &6
MOVL(498) &0 MEMORY_6
LD TR0
AND=(300) STACK_LOC &7
MOVL(498) &0 MEMORY_7
LD TR0
AND=(300) STACK_LOC &8
MOVL(498) &0 MEMORY_8
LD TR0
AND=(300) STACK_LOC &9
MOVL(498) &0 MEMORY_9
LD TR0
AND=(300) STACK_LOC &10
MOVL(498) &0 MEMORY_10
LD TR0
AND=(300) STACK_LOC &11
MOVL(498) &0 MEMORY_11
LD TR0
AND=(300) STACK_LOC &12
MOVL(498) &0 MEMORY_12
LD TR0
AND=(300) STACK_LOC &13
MOVL(498) &0 MEMORY_13
LD TR0
AND=(300) STACK_LOC &14
MOVL(498) &0 MEMORY_14
LD TR0
AND=(300) STACK_LOC &15
MOVL(498) &0 MEMORY_15
LD TR0
AND=(300) STACK_LOC &16
MOVL(498) &0 MEMORY_16
LD TR0
AND=(300) STACK_LOC &17
MOVL(498) &0 MEMORY_17
LD TR0
AND=(300) STACK_LOC &18
MOVL(498) &0 MEMORY_18
LD TR0
AND=(300) STACK_LOC &19
MOVL(498) &0 MEMORY_19
LD TR0
AND=(300) STACK_LOC &20
MOVL(498) &0 MEMORY_20
LD TR0
AND=(300) STACK_LOC &21
MOVL(498) &0 MEMORY_21
LD TR0
AND=(300) STACK_LOC &22
MOVL(498) &0 MEMORY_22
LD TR0
AND=(300) STACK_LOC &23
MOVL(498) &0 MEMORY_23
LD TR0
AND=(300) STACK_LOC &24
MOVL(498) &0 MEMORY_24
LD TR0
AND=(300) STACK_LOC &25
MOVL(498) &0 MEMORY_25
LD TR0
AND=(300) STACK_LOC &26
MOVL(498) &0 MEMORY_26
LD TR0
AND=(300) STACK_LOC &27
MOVL(498) &0 MEMORY_27
LD TR0
AND=(300) STACK_LOC &28
MOVL(498) &0 MEMORY_28
LD TR0
AND=(300) STACK_LOC &29
MOVL(498) &0 MEMORY_29
LD TR0
AND=(300) STACK_LOC &30
MOVL(498) &0 MEMORY_30
LD TR0
AND=(300) STACK_LOC &31
MOVL(498) &0 MEMORY_31
LD TR0
AND=(300) STACK_LOC &32
MOVL(498) &0 MEMORY_32
LD TR0
AND=(300) STACK_LOC &33
MOVL(498) &0 MEMORY_33
LD TR0
AND=(300) STACK_LOC &34
MOVL(498) &0 MEMORY_34
LD TR0
AND=(300) STACK_LOC &35
MOVL(498) &0 MEMORY_35
LD TR0
AND=(300) STACK_LOC &36
MOVL(498) &0 MEMORY_36
LD TR0
AND=(300) STACK_LOC &37
MOVL(498) &0 MEMORY_37
LD TR0
AND=(300) STACK_LOC &38
MOVL(498) &0 MEMORY_38
LD TR0
AND=(300) STACK_LOC &39
MOVL(498) &0 MEMORY_39
LD TR0
AND=(300) STACK_LOC &40
MOVL(498) &0 MEMORY_40
LD TR0
AND=(300) STACK_LOC &41
MOVL(498) &0 MEMORY_41
LD TR0
AND=(300) STACK_LOC &42
MOVL(498) &0 MEMORY_42
LD TR0
AND=(300) STACK_LOC &43
MOVL(498) &0 MEMORY_43
LD TR0
AND=(300) STACK_LOC &44
MOVL(498) &0 MEMORY_44
LD TR0
AND=(300) STACK_LOC &45
MOVL(498) &0 MEMORY_45
LD TR0
AND=(300) STACK_LOC &46
MOVL(498) &0 MEMORY_46
LD TR0
AND=(300) STACK_LOC &47
MOVL(498) &0 MEMORY_47
LD TR0
AND=(300) STACK_LOC &48
MOVL(498) &0 MEMORY_48
LD TR0
AND=(300) STACK_LOC &49
MOVL(498) &0 MEMORY_49
LD TR0
AND=(300) STACK_LOC &50
MOVL(498) &0 MEMORY_50

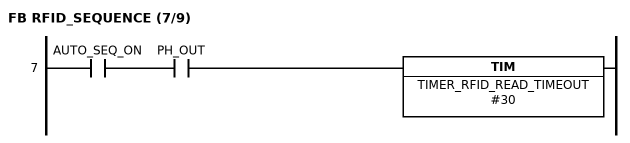
; rung 7
LD AUTO_SEQ_ON
AND PH_OUT
TIM TIMER_RFID_READ_TIMEOUT #30

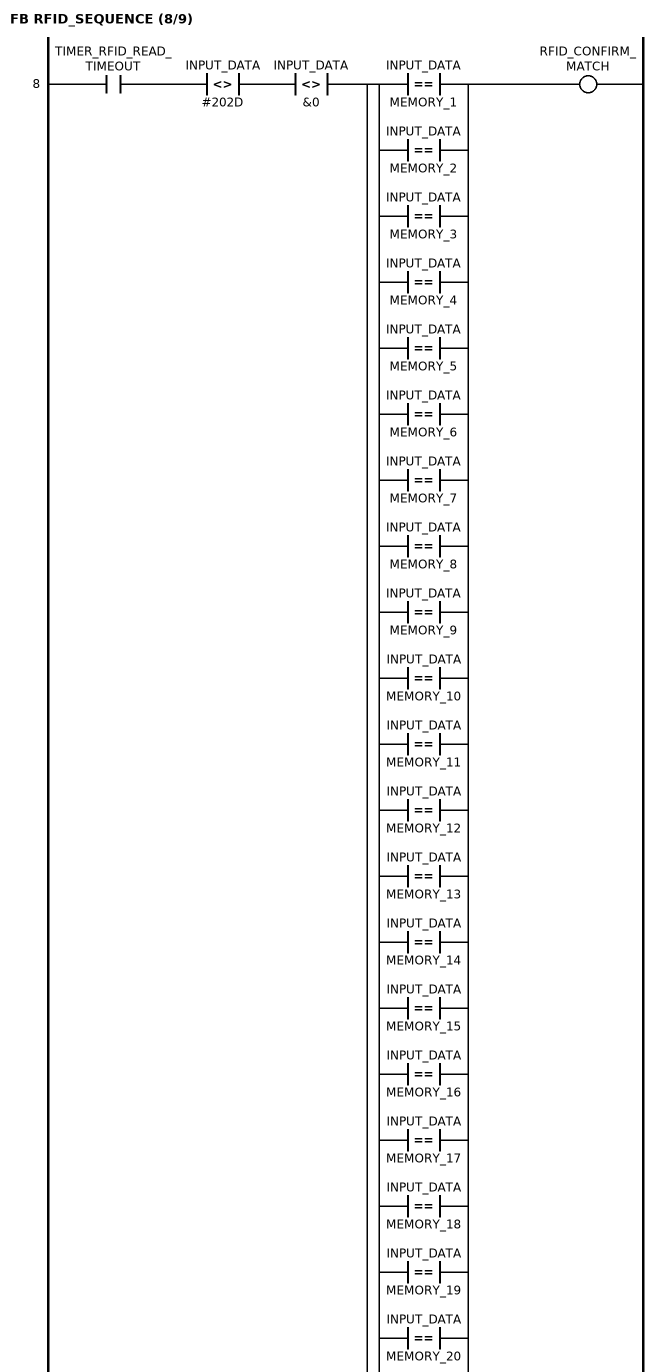

